// TIA Portal project "Schrittmotor" (V14)

(* hardware
DEVICE "S7-1200-Station_1"  S7-1200 Station
   slot 0: "Baugruppenträger_0"  Rack  V1.0
   slot 1: "PLC"  CPU 1214C DC/DC/DC  6ES7 214-1AG40-0XB0  V4.1
   slot 3: "AQ 1x12BIT_1"  6ES7 232-4HA30-0XB0  V1.0
DEVICE "HMI"  KTP700 Basic PN
   slot 0: "HMI"  HMI  6AV2 123-2GB03-0AX0  13.0.1.0
   slot 1: "HMI_RT_1"  KTP700 Basic PN  6AV2 123-2GB03-0AX0  13.0.1.0
   slot 5: "HMI.IE_CP_1"  PROFINET Schnittstelle
      slot 1: "PROFINET Schnittstelle_1"  PROFINET Schnittstelle
         slot 1: "Port_1"  Port
*)

// ===== PLC "PLC"  CPU 1214C DC/DC/DC =====

VAR_GLOBAL   // PLC tag table "Standard-Variablentabelle"
   "System_Byte" AT %MB100 : Byte;
   "FirstScan" AT %M100.0 : Bool;
   "DiagStatusUpdate" AT %M100.1 : Bool;
   "AlwaysTRUE" AT %M100.2 : Bool;
   "AlwaysFALSE" AT %M100.3 : Bool;
   "Clock_Byte" AT %MB110 : Byte;
   "Clock_10Hz" AT %M110.0 : Bool;
   "Clock_5Hz" AT %M110.1 : Bool;
   "Clock_2.5Hz" AT %M110.2 : Bool;
   "Clock_2Hz" AT %M110.3 : Bool;
   "Clock_1.25Hz" AT %M110.4 : Bool;
   "Clock_1Hz" AT %M110.5 : Bool;
   "Clock_0.625Hz" AT %M110.6 : Bool;
   "Clock_0.5Hz" AT %M110.7 : Bool;
   "A" AT %Q0.0 : Bool;   // Wicklungsanschluss A
   "A\" AT %Q0.1 : Bool;   // Wicklungsanschluss A\
   "B" AT %Q0.2 : Bool;   // Wicklungsanschluss B
   "B\" AT %Q0.3 : Bool;   // Wicklungsanschluss B\
   "Motorposition_Ist" AT %MW10 : Int;   // Motorposition Istwert
   "Motorposition_Soll" AT %MW12 : Int;   // Motorposition Sollwert
   "Motor_Start" AT %M20.0 : Bool;   // Motor Start
   "Motor_Stop" AT %M20.1 : Bool;   // Motor Stop
   "AlleAusgänge" AT %QW0 : Word;
END_VAR

FUNCTION "fcSchrittmotor" : Void   // FC1, FBD
{ S7_Optimized_Access := 'TRUE' }
VERSION : 0.1
BEGIN
END_FUNCTION

ORGANIZATION_BLOCK "Main"   // OB1, LAD, ProgramCycle
TITLE = "Main Program Sweep (Cycle)"
{ S7_Optimized_Access := 'TRUE' }
VERSION : 0.1
   VAR_INPUT
      Initial_Call : Bool;   // Initial call of this OB
      Remanence : Bool;   // =True, if remanent data are available
   END_VAR
BEGIN

REGION Network 1: -Q1
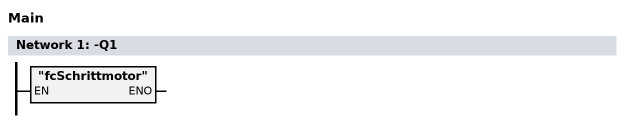
   RUNG wire#powerrail
      "fcSchrittmotor"()
   END_RUNG
   // the same network as SCL:
   "fcSchrittmotor"();
END_REGION
END_ORGANIZATION_BLOCK

ORGANIZATION_BLOCK "Startup"   // OB100, SCL, Startup
TITLE = "Complete Restart"
{ S7_Optimized_Access := 'TRUE' }
VERSION : 0.1
   VAR_INPUT
      LostRetentive : Bool;   // True if retentive data are lost
      LostRTC : Bool;   // True if date and time are lost
   END_VAR
BEGIN
   "AlleAusgänge" := 16#0000;
END_ORGANIZATION_BLOCK

(* ===== HMI "HMI_RT_1" =====
connection "HMI_Verbindung_1": ETHERNET, SMART_S7_1200_OMS

HMI tags "Standard-Variablentabelle"
   "MotorPosition_Ist" : Int = PLC Motorposition_Ist AT %MW10, 1 s
   "MotorPosition_Soll" : Int = PLC Motorposition_Soll AT %MW12, 1 s
   "Motor_Start" : Bool = PLC Motor_Start AT %M20.0, 1 s
   "Motor_Stop" : Bool = PLC Motor_Stop AT %M20.1, 1 s

screen "SchrittMotor" 800x480
   IOField "EA-Feld_1" at 566,107 size 96x32; FormatPattern 9999999
   Switch "Schalter_1" at 567,163 size 64x32; CaptionText 'Switch'; TextOff 'OFF'; TextOn 'ON'
*)